FUNCTION_BLOCK SpacerRecollectionUnit //EXTENDS SectionEx
VAR_IN_OUT
	robot : RobotA26;
	robotSlider : ServoNC;
END_VAR
VAR_INPUT
	conveyorOccupied_A24_LRC_C01 : BOOL;
	conveyorOccupied_A24_LRC_C03 : BOOL;
	conveyorOccupied_A24_LRC_C05 : BOOL;
	conveyorOccupied_A24_LRC_C07 : BOOL;
	conveyorOccupied_A24_LRC_C09 : BOOL;
	conveyorOccupied_A24_LRC_C11 : BOOL;
	conveyorOccupied_A24_LRC_C13 : BOOL;
	
	spacerPresent_A24_LRC_C02 : BOOL;
	spacerPresent_A24_LRC_C04 : BOOL;
	spacerPresent_A24_LRC_C06 : BOOL;
	spacerPresent_A24_LRC_C08 : BOOL;
	spacerPresent_A24_LRC_C10 : BOOL;
	spacerPresent_A24_LRC_C12 : BOOL;
END_VAR
VAR_OUTPUT
	ready : BOOL;
	busy : BOOL;
	done : BOOL;
	error : BOOL;
	
	failCounter : INT;
END_VAR
VAR
	step : (IDLE, SLIDE, PICK_SPACER, COMPLETE);
	iPosition : INT;
END_VAR
VAR //slider positions
	pickPos1, pickPos2 : LREAL;
END_VAR

ready := step = 0;
busy := step > 0;
done := done;
error := error;

IF 
	conveyorOccupied_A24_LRC_C01 OR
	conveyorOccupied_A24_LRC_C03 OR
	conveyorOccupied_A24_LRC_C05 OR
	conveyorOccupied_A24_LRC_C07 OR
	conveyorOccupied_A24_LRC_C09 OR
	conveyorOccupied_A24_LRC_C11 OR
	conveyorOccupied_A24_LRC_C13
THEN
	robot.clearCommand();
	
ELSE
	//remove spacers from transfer conveyors in ascending order
	process();
	
END_IF

METHOD process : BOOL
VAR
	spacersPresent : ARRAY[1..6] OF BOOL := [
		spacerPresent_A24_LRC_C02,
		spacerPresent_A24_LRC_C04,
		spacerPresent_A24_LRC_C06,
		spacerPresent_A24_LRC_C08,
		spacerPresent_A24_LRC_C10,
		spacerPresent_A24_LRC_C12];
END_VAR
VAR CONSTANT
	suctionDistance : INT := 10;
END_VAR
{warning disable C0371}

iPosition := MAX(1, iPosition); //value is always at least 1

CASE step OF
	IDLE:
		IF DataIsEmpty(arr := ADR(spacersPresent), arrSize := SIZEOF(spacersPresent)) THEN
			robotSlider.toHome();
			
			iPosition := 0;
			failCounter := 0;
			process := TRUE;
		
		ELSIF NOT spacersPresent[iPosition] THEN
			iPosition := iPosition + 1;
			
		ELSIF robot.Ready THEN
			step := SLIDE;
		END_IF
		
	SLIDE:
		CASE iPosition OF
			1,2,3:		robotSlider.moveAbsolute(newTarget := pickPos1);
			4,5,6:		robotSlider.moveAbsolute(newTarget := pickPos2);
		END_CASE
		
		//replace this condition with WithinTolerance() if the slider spends too long adjusting its position
		IF robotSlider.CurrentPosition = robotSlider.TargetPosition THEN
			step := PICK_SPACER;
		END_IF
		
	PICK_SPACER:		
		IF robot.eoatDistance > suctionDistance THEN
			robot.HoldMaterial := 'SPACER';
		ELSE
			robot.HoldMaterial := '';
		END_IF
	
		IF robot.Done THEN
			step := COMPLETE;
		ELSE
			robot.setGroup(group := 1, value := TaskA26.PICK_SPACER);
			robot.setGroup(group := 2, value := iPosition);
		END_IF
		
	COMPLETE:
		robot.HoldMaterial := '';
		
		IF spacersPresent[iPosition] THEN
			failCounter := failCounter + 1;
		END_IF
		
		robot.clearCommand();
		step := 0;
	
END_CASE
END_METHOD

END_FUNCTION_BLOCK

(* stored: Version 1.1.0.1, ProductVersion 3.1.4024.11
   POU SpacerRecollectionUnit: Id {6fea2dc6-ce06-4fa1-9588-ba3bbddda180}, SpecialFunc None
   Method process: Id {0707ef1b-9ba5-4d26-b34d-69bdd29b3450} *)
